TYPE "MatCountPersistent"
VERSION : 0.1
// Block: MatCountPersistent
   STRUCT
      Data : MatCountData;
      Par : MatCountPar;
   END_STRUCT;

END_TYPE
